// TIA Portal V17 export
// export: Created 2024-08-09T12:53:16.2339807Z, ExportSetting WithDefaults, DisplayName Totally Integrated Automation Portal, DisplayVersion V17 Update 7, DisplayName TIA Portal Openness, DisplayVersion V17 Update 7, DisplayName TIA Portal Version Control Interface, DisplayVersion V17, DisplayName STEP 7 Professional, DisplayVersion V17 Update 7, DisplayName STEP 7 Safety, DisplayVersion V17 Update 6, DisplayName WinCC Professional, DisplayVersion V17 Update 7
TYPE "S_D_IO"
TITLE = Structure pour les entrees sorties digitales
// Constitution de la structure des entrees sorties
// stored: IsFailsafeCompliant false
   STRUCT
      Tps_Picke { ExternalAccessible := 'False'; ExternalVisible := 'False'; ExternalWritable := 'False'} : Date_And_Time;   // Le prelevement du temps pour les filtres
      Filtr_0_1 : Time := T#100MS;   // temps de filtrage passage de l'IO de false a true
      Filtr_1_0 : Time := T#100MS;   // temps de filtrage passage de l'IO de true a false
      Description : String[100];   // Description de l'IO
      Mnemonique : String[20];   // Mnemonique du mobile
      Reseau : USInt;   // Le reseau ou se trouve cette entree/sortie
      Rack : USInt;   // Le rack ou cette entree/sortie est montee
      Carte : USInt;   // La carte ou cette entree/sortie est cablee
      Type_IO { ExternalAccessible := 'False'; ExternalVisible := 'False'; ExternalWritable := 'False'} : Char;   // Type dde l'IO si Entree = 'E' si sortie = 'S'
      Log_Nc : Bool;   // logique de l'entree false = NO, True = NC
      Masque : Bool;   // Cette entree est elle masquee
      Force : Bool;   // Forcage de cette entree/sortie
      Etat : Bool;   // Etat de sortie de l'IO
      Adr_IO : Bool;   // L'adresse de cette entree/sortie
      Init_Tps_Filtre { ExternalAccessible := 'False'; ExternalVisible := 'False'; ExternalWritable := 'False'} : Bool;
   END_STRUCT;
END_TYPE
